TYPE ST_LineDataParCmd :
STRUCT
    Reserved : BOOL; // line data takes no command: physical four-structure contract
END_STRUCT
END_TYPE

(* stored: Version 1.1.0.1, ProductVersion 3.1.4024.12
   DUT ST_LineDataParCmd: Id {a9619897-94e4-4830-9f6d-dff2ea1a8d39} *)
